# EPICS autosave request: kinetixApp/Db/kinetix_settings.req
file "ADBase_settings.req", P=$(P), R=$(R)
